# EPICS autosave request: iocBoot/ioc13idb_ps1/auto_settings.req
file "vimba_settings.req",          P=$(P),  R=cam1:
file "NDStdArrays_settings.req",    P=$(P),  R=image1:
file "commonPlugin_settings.req",   P=$(P)
